// Writes an enum value, without a tag, to the stream.
FUNCTION F_WriteEnum : HRESULT
VAR_IN_OUT      
    stCtx : ST_WriteContext;
END_VAR
VAR_INPUT
    nValue : DINT;
END_VAR
VAR
END_VAR


F_WriteEnum := F_WriteInt32(stCtx, nValue);

END_FUNCTION

(* stored: Version 1.1.0.1
   POU F_WriteEnum: Id {9efd0922-0421-488b-8db4-fa01c76f70a4}, SpecialFunc None *)
